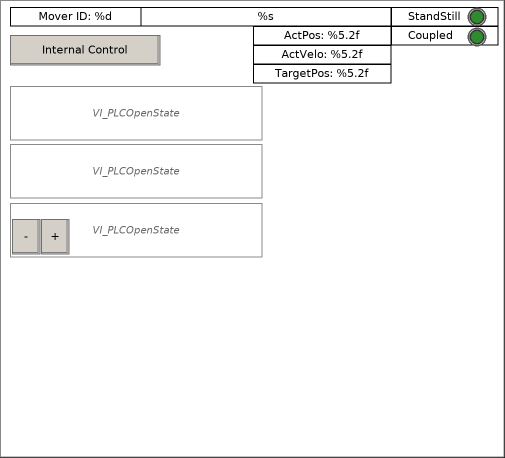
VISUALIZATION VI_MoverVisu  // 505x458
VAR_IN_OUT
	fbMover : FB_Mover;
END_VAR
    Rectangle (0,0 505x458)
    Rectangle (140,7 251x19), "%s", text variable: fbMover.ax.Status.MotionState, text list: 'AxisState_txt'
    Frame (10,86 252x54)
        shows VI_PLCOpenState(bExecute := fbMover.fbPower.Enable, sName := 'Power', bBusy := fbMover.fbPower.Busy, bDone := fbMover.fbPower.Status, bError := fbMover.fbPower.Error, bCommandAborted := fbMover.bTmp, ErrorID := fbMover.fbPower.ErrorID)
    Frame (10,144 252x54)
        shows VI_PLCOpenState(bExecute := fbMover.fbReset.Execute, sName := 'Reset', bBusy := fbMover.fbReset.Busy, bDone := fbMover.fbReset.Done, bError := fbMover.fbReset.Error, bCommandAborted := fbMover.bTmp, ErrorID := fbMover.fbReset.ErrorId)
    Button (10,35 150x30), "Internal Control", tooltip "Enable Visu Control, all methods will be locked"
        toggle fbMover.bInternalControl
    Rectangle (391,7 107x19), "StandStill"
    Lamp1 (466,6 22x22), variable: fbMover.ax.Status.StandStill, style: Lamp-Lamp1-Green
    Rectangle (10,7 131x19), "Mover ID: %d", text variable: fbMover.udiID
    Rectangle (253,26 138x19), "ActPos: %5.2f", text variable: fbMover.ax.NcToPlc.ModuloActPos, text list: 'AxisState_txt'
    Rectangle (253,45 138x19), "ActVelo: %5.2f", text variable: fbMover.ax.NcToPlc.ActVelo, text list: 'AxisState_txt'
    Rectangle (391,26 107x19), "Coupled"
    Lamp1 (466,26 22x22), variable: fbMover.ax.Status.Coupled, style: Lamp-Lamp1-Green
    Frame (10,203 252x54)
        shows VI_PLCOpenState(bExecute := fbMover.bTmp, sName := 'JogCA', bBusy := fbMover.fbJogCA.Busy, bDone := fbMover.fbJogCA.Done, bError := fbMover.fbJogCA.Error, bCommandAborted := fbMover.fbJogCA.CommandAborted, ErrorID := fbMover.fbJogCA.ErrorID)
    Button (12,219 28x35), "-"
        toggle fbMover.fbJogCA.JogBackwards
    Button (41,219 28x35), "+"
        toggle fbMover.fbJogCA.JogForward
    Rectangle (253,64 138x19), "TargetPos: %5.2f", text variable: fbMover.lrTargetPos, text list: 'AxisState_txt'
END_VISUALIZATION

(* stored: Version 1.1.0.1, ProductVersion 3.1.4024.11
   Visu VI_MoverVisu: Id {48a3d2e5-a95b-4bd1-99f5-575a625732f7} *)
